SUBAPPLICATION GreenWhiteBackground1SC (* Hintergrundfarbe (TRUE -> Grün, FALSE -> Weiß) für 1 Objekt (Kompakt) *)
  (* Standard: 61499-2 *)
  (* Version 1.0, 2024-01-01, franz *)
  PACKAGE MyLib::sys;
  IMPORT isobus::UT::Q::const::IDs::ID_NULL;
  IMPORT isobus::UT::Q::types::s1ObjectID;
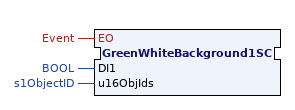
  EVENT_INPUT
    EO;
  END_EVENT
  VAR_INPUT
    DI1 : BOOL; (* Selector *)
    u16ObjIds : isobus::UT::Q::types::s1ObjectID := (u16ObjId := ID_NULL); (* Object IDs *)
  END_VAR
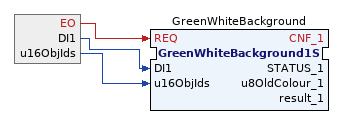
  SUBAPPS
    GreenWhiteBackground : MyLib::sys::GreenWhiteBackground1S;
  END_SUBAPPS
  EVENT_CONNECTIONS
    EO TO GreenWhiteBackground.REQ;
  END_CONNECTIONS
  DATA_CONNECTIONS
    u16ObjIds TO GreenWhiteBackground.u16ObjIds;
    DI1 TO GreenWhiteBackground.DI1;
  END_CONNECTIONS
END_SUBAPPLICATION
